# EPICS alarm handler configuration: mps_database/bare/alarms/areas/mpln_undh_mp04.alhConfig
GROUP NULL MPLN:UNDH:MP04:1
$ALIAS MPS Link Node 139
$GUIDANCE
LTUH MPS
   Group Name: MPLN:UNDH:MP04:1
   Summary PV:  MPLN:UNDH:MP04:1:STATSUMY
$END
CHANNEL  MPLN:UNDH:MP04:1    MPLN:UNDH:MP04:1:MPS_EN_RBV		-----
CHANNEL  MPLN:UNDH:MP04:1    MPLN:UNDH:MP04:1:LC1_MODE_RBV		-----
